Fanuc KAREL source: POS_REG_TYPE.kl

PROGRAM T
%NOLOCKGROUP
VAR
 v0 : INTEGER
 v1 : INTEGER
 v2 : INTEGER
 v3 : INTEGER
 v4 : INTEGER
BEGIN
 POS_REG_TYPE(v0, v1, v2, v3, v4)
END T
